KUKA KRL program: ps_603geo_x1.src, ps_603geo_x1.dat

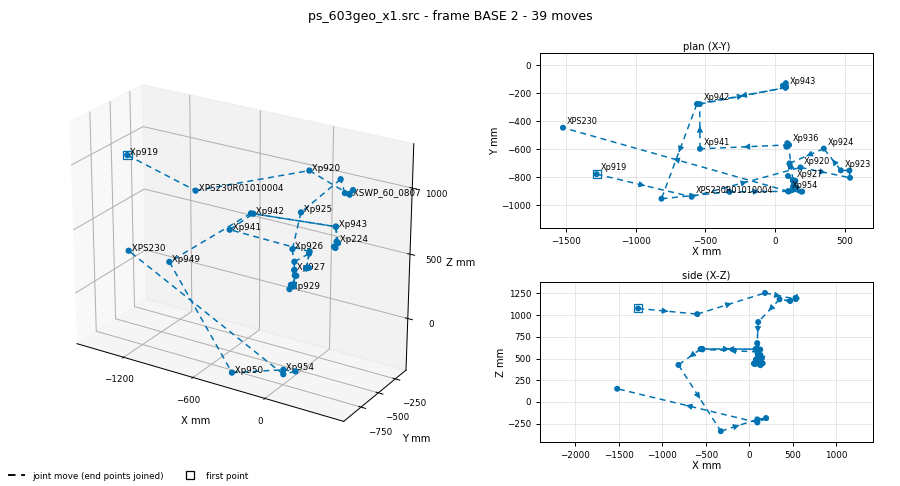
[picture p0: tool path of ps_603geo_x1.src in frame BASE 2, 39 of 39 moves have a stored position in this frame; points joined in program order, loops and branches not executed]
--- ps_603geo_x1.src ---
&ACCESS RV2
&REL 97
&COMMENT Solda Geometria x1
DEF ps_603geo_x1( )
EXT e_Fraes2 ( )
EXT f_Fraes2 ( )

  ;FOLD INI;%{PE}%V2.2.2,%MKUKATPBASIS,%CINIT,%VCOMMON,%P
  ;FOLD BAS INI;%{PE}%V2.2.2,%MKUKATPBASIS,%CINIT,%VINIT,%P
  INTERRUPT DECL 3 WHEN $STOPMESS==TRUE DO IR_STOPM ( )
  INTERRUPT ON 3
  BAS (#INITMOV,0 )
  ;ENDFOLD
  ;FOLD A20 INI;%{E}%V2.2.2,%MKUKATPA20,%CINIT,%VINIT,%P
  IF ARC20==TRUE THEN
    A20 (ARC_INI)
    INTERRUPT DECL 6 WHEN $CYCFLAG[3]==FALSE DO A20(TECH_STOP2)
  ENDIF
  ;ENDFOLD
  ;FOLD A10 INI;%{E}%V2.2.2,%MKUKATPARC,%CINIT,%VINIT,%P
  IF A10_OPTION==#ACTIVE THEN
    INTERRUPT DECL 4 WHEN $CYCFLAG[2]==FALSE DO A10 (#APPL_ERROR)
    INTERRUPT DECL 7 WHEN A_ARC_SWI==#ACTIVE DO A10 (#ARC_SEAM)
    INTERRUPT DECL 5 WHEN A_FLY_ARC==TRUE DO A10 (#HPU_ARC)
    INTERRUPT  ON 5
    A10_INI ( )
  ENDIF
  ;ENDFOLD
  ;FOLD GRIPPER INI;%{E}%V2.2.2,%MKUKATPGRIPPER,%CINIT,%VINIT,%P
  USER_GRP(0,DUMMY,DUMMY,GDEFAULT)
  ;ENDFOLD
  ;FOLD SPOT INI;%{E}%V.2.2,%MKUKATPSPOT,%CINIT,%VINIT,%P
  USERSPOT(#INIT)
  ;ENDFOLD
  ;FOLD TOUCHSENSE INI;%{E}%V2.2.2,%MKUKATPTS,%CINIT,%VINIT,%P
  IF H70_OPTION THEN
    INTERRUPT DECL 15 WHEN $MEAS_PULSE[TOUCH_I[TOUCH_ACTIVE].IN_NR] DO H70 (6,CD0 )
    INTERRUPT DECL 16 WHEN $ZERO_MOVE DO H70 (7,CD0 )
    INTERRUPT DECL 17 WHEN $TECHPAR_C[FG_TOUCH,8]>0.5 DO H70 (8,CD0)
    H70 (1,CD0 )
  ENDIF
  ;ENDFOLD
  ;FOLD USER INI;%{P}%V2.2.2,%MKUKATPUSER,%CINIT,%VINIT,%P
  ;Make your modifications here
  ;ENDFOLD
  ;ENDFOLD

; Caracterização dos meios de produção:
; Versão Atual:
; 19/07/2013 12:00 Name: P13.060-R3 CHANGES: Solda Geometria X1
; Accelo

chk_w2_wechs_ok ( )        ;VERIFICAÇÃO DE FERRAMENTA: x1

IF (NOT(GHOST())) THEN
IF MaxStandMenge(2) THEN
  MaxStandmengeErreicht(2)
ENDIF

IF Elektrodenwechsel(2) THEN
  e_Fraes2()                  ; Fresa Pinca X1
ENDIF
ENDIF

;FOLD PTP p919  Vel= 100 % P_OLP1 Tool[2]:Gun X1                   Base[2]:Accelo;%{PE}%R 4.1.16,%MKUKATPBASIS,%CMOVE,%VPTP,%P 1:PTP, 2:p919, 3:, 5:100, 7:P_OLP1
$BWDSTART = FALSE
PDAT_ACT=PP_OLP1
BAS(#PTP_DAT)
FDAT_ACT=Fp919
BAS(#FRAMES)
BAS(#VEL_PTP,100)
PTP Xp919
;ENDFOLD

;FOLD ; START INTERLOCK 2 COM R4;%{PE}%R2.2,%MKUKATPBASIS,%CCOMMENT,%VNORMAL,%P 2: START INTERLOCK 2 COM R4
;ENDFOLD
;FOLD Kollision.Ueberwachung_4_Ein ;%{PE}%MKUKATPUSER
COLLSTOP( 4, 1 ) ;INTERRUPTUEBERWACHT
;ENDFOLD

;FOLD PTP PS230R01010004 CONT Vel= 100 % PDAT3 Tool[2]:Gun X1                   Base[2]:Accelo;%{PE}%R 4.1.16,%MKUKATPBASIS,%CMOVE,%VPTP,%P 1:PTP, 2:PS230R01010004, 3:C_PTP, 5:100, 7:PDAT3
$BWDSTART = FALSE
PDAT_ACT=PPDAT3
BAS(#PTP_DAT)
FDAT_ACT=FPS230R01010004
BAS(#FRAMES)
BAS(#VEL_PTP,100)
PTP XPS230R01010004 C_PTP
;ENDFOLD

;FOLD OUT 839 'Soldando'  State= TRUE ;%{PE}%R 4.1.16,%MKUKATPBASIS,%COUT,%VOUTX,%P 2:839, 3:'Soldando', 5:TRUE, 6:
$OUT[839]=TRUE
;ENDFOLD
;FOLD OUT 848 'Area de Solda'  State= FALSE ;%{PE}%R 4.1.16,%MKUKATPBASIS,%COUT,%VOUTX,%P 2:848, 3:'Area de Solda', 5:FALSE, 6:
$OUT[848]=FALSE
;ENDFOLD

;FOLD PTP p920 CONT Vel= 100 % P_OLP2 Tool[2]:Gun X1                   Base[2]:Accelo;%{PE}%R 4.1.16,%MKUKATPBASIS,%CMOVE,%VPTP,%P 1:PTP, 2:p920, 3:C_PTP, 5:100, 7:P_OLP2
$BWDSTART = FALSE
PDAT_ACT=PP_OLP2
BAS(#PTP_DAT)
FDAT_ACT=Fp920
BAS(#FRAMES)
BAS(#VEL_PTP,100)
PTP Xp920 C_PTP
;ENDFOLD

;FOLD ; SWP_60_0807;%{PE}%R2.2,%MKUKATPBASIS,%CCOMMENT,%VNORMAL,%P 2: SWP_60_0807
;ENDFOLD
;FOLD PTP SWP_60_0807 PDAT4 SPOT Gun= 2 RETR CLS PgNo1= 121 ACTIVE= 1 Tool[2]:Gun X1                   Base[2]:Accelo;%{PE}%R 4.1.12,%MKUKATPSPOT,%CSPOT,%VPTP,%P 1:PTP, 2:SWP_60_0807, 3:, 5:100, 7:PDAT4, 10:2, 12:#FIRST, 14:#CLO, 16:121, 18:1, 20:0, 22:0, 24:1, 25:NORMAL
$BWDSTART = FALSE
PDAT_ACT=PPDAT4
BAS(#PTP_DAT)
FDAT_ACT=FSWP_60_0807
BAS(#FRAMES)
BAS(#VEL_PTP,PPDAT4.VEL)
S_ACT.GUN=2
S_ACT.PAIR=SDEFAULT.PAIR
S_ACT.RETR=#CLO
S_ACT.CLO_TM=1
S_ACT.PGNO1=121
S_ACT.PGNO2=SDEFAULT.PGNO2
S_ACT.PRESS1=SDEFAULT.PRESS1
S_ACT.PRESS2=SDEFAULT.PRESS2
S_READY=FALSE
PTP XSWP_60_0807
USERSPOT(#SPOT, S_ACT)
WAIT FOR S_READY
;ENDFOLD

;FOLD ; SWP_60_0403;%{PE}%R2.2,%MKUKATPBASIS,%CCOMMENT,%VNORMAL,%P 2: SWP_60_0403
;ENDFOLD
;FOLD PTP SWP_60_0403 PDAT5 SPOT Gun= 2 RETR OPN PgNo1= 122 ACTIVE= 1 Tool[2]:Gun X1                   Base[2]:Accelo;%{PE}%R 4.1.12,%MKUKATPSPOT,%CSPOT,%VPTP,%P 1:PTP, 2:SWP_60_0403, 3:, 5:100, 7:PDAT5, 10:2, 12:#FIRST, 14:#OPN, 16:122, 18:1, 20:0, 22:0, 24:1, 25:NORMAL
$BWDSTART = FALSE
PDAT_ACT=PPDAT5
BAS(#PTP_DAT)
FDAT_ACT=FSWP_60_0403
BAS(#FRAMES)
BAS(#VEL_PTP,PPDAT5.VEL)
S_ACT.GUN=2
S_ACT.PAIR=SDEFAULT.PAIR
S_ACT.RETR=#OPN
S_ACT.CLO_TM=1
S_ACT.PGNO1=122
S_ACT.PGNO2=SDEFAULT.PGNO2
S_ACT.PRESS1=SDEFAULT.PRESS1
S_ACT.PRESS2=SDEFAULT.PRESS2
S_READY=FALSE
PTP XSWP_60_0403
USERSPOT(#SPOT, S_ACT)
WAIT FOR S_READY
;ENDFOLD

;FOLD PTP p923 CONT Vel= 100 % P_OLP5 Tool[2]:Gun X1                   Base[2]:Accelo;%{PE}%R 4.1.16,%MKUKATPBASIS,%CMOVE,%VPTP,%P 1:PTP, 2:p923, 3:C_PTP, 5:100, 7:P_OLP5
$BWDSTART = FALSE
PDAT_ACT=PP_OLP5
BAS(#PTP_DAT)
FDAT_ACT=Fp923
BAS(#FRAMES)
BAS(#VEL_PTP,100)
PTP Xp923 C_PTP
;ENDFOLD
;FOLD PTP p924 CONT Vel= 100 % P_OLP6 Tool[2]:Gun X1                   Base[2]:Accelo;%{PE}%R 4.1.16,%MKUKATPBASIS,%CMOVE,%VPTP,%P 1:PTP, 2:p924, 3:C_PTP, 5:100, 7:P_OLP6
$BWDSTART = FALSE
PDAT_ACT=PP_OLP6
BAS(#PTP_DAT)
FDAT_ACT=Fp924
BAS(#FRAMES)
BAS(#VEL_PTP,100)
PTP Xp924 C_PTP
;ENDFOLD
;FOLD PTP p925 CONT Vel= 100 % P_OLP7 Tool[2]:Gun X1                   Base[2]:Accelo;%{PE}%R 4.1.16,%MKUKATPBASIS,%CMOVE,%VPTP,%P 1:PTP, 2:p925, 3:C_PTP, 5:100, 7:P_OLP7
$BWDSTART = FALSE
PDAT_ACT=PP_OLP7
BAS(#PTP_DAT)
FDAT_ACT=Fp925
BAS(#FRAMES)
BAS(#VEL_PTP,100)
PTP Xp925 C_PTP
;ENDFOLD
;FOLD PTP p926 CONT Vel= 100 % P_OLP8 Tool[2]:Gun X1                   Base[2]:Accelo;%{PE}%R 4.1.16,%MKUKATPBASIS,%CMOVE,%VPTP,%P 1:PTP, 2:p926, 3:C_PTP, 5:100, 7:P_OLP8
$BWDSTART = FALSE
PDAT_ACT=PP_OLP8
BAS(#PTP_DAT)
FDAT_ACT=Fp926
BAS(#FRAMES)
BAS(#VEL_PTP,100)
PTP Xp926 C_PTP
;ENDFOLD

;FOLD ; END INTERLOCK 2 COM R4;%{PE}%R2.2,%MKUKATPBASIS,%CCOMMENT,%VNORMAL,%P 2: END INTERLOCK 2 COM R4
;ENDFOLD
;FOLD Kollision.Ueberwachung_4_Aus ;%{PE}%MKUKATPUSER
COLLSTOP( 4, 2 )
;ENDFOLD

;FOLD PTP p927 CONT Vel= 100 % P_OLP9 Tool[2]:Gun X1                   Base[2]:Accelo;%{PE}%R 4.1.16,%MKUKATPBASIS,%CMOVE,%VPTP,%P 1:PTP, 2:p927, 3:C_PTP, 5:100, 7:P_OLP9
$BWDSTART = FALSE
PDAT_ACT=PP_OLP9
BAS(#PTP_DAT)
FDAT_ACT=Fp927
BAS(#FRAMES)
BAS(#VEL_PTP,100)
PTP Xp927 C_PTP
;ENDFOLD
;FOLD PTP p928 CONT Vel= 100 % P_OLP10 Tool[2]:Gun X1                   Base[2]:Accelo;%{PE}%R 4.1.16,%MKUKATPBASIS,%CMOVE,%VPTP,%P 1:PTP, 2:p928, 3:C_PTP, 5:100, 7:P_OLP10
$BWDSTART = FALSE
PDAT_ACT=PP_OLP10
BAS(#PTP_DAT)
FDAT_ACT=Fp928
BAS(#FRAMES)
BAS(#VEL_PTP,100)
PTP Xp928 C_PTP
;ENDFOLD
;FOLD PTP p929 CONT Vel= 100 % P_OLP11 Tool[2]:Gun X1                   Base[2]:Accelo;%{PE}%R 4.1.16,%MKUKATPBASIS,%CMOVE,%VPTP,%P 1:PTP, 2:p929, 3:C_PTP, 5:100, 7:P_OLP11
$BWDSTART = FALSE
PDAT_ACT=PP_OLP11
BAS(#PTP_DAT)
FDAT_ACT=Fp929
BAS(#FRAMES)
BAS(#VEL_PTP,100)
PTP Xp929 C_PTP
;ENDFOLD

;FOLD ; SWP_60_0769;%{PE}%R2.2,%MKUKATPBASIS,%CCOMMENT,%VNORMAL,%P 2: SWP_60_0769
;ENDFOLD
;FOLD PTP SWP_60_0769 PDAT6 SPOT Gun= 2 RETR OPN PgNo1= 123 ACTIVE= 1 Tool[2]:Gun X1                   Base[2]:Accelo;%{PE}%R 4.1.12,%MKUKATPSPOT,%CSPOT,%VPTP,%P 1:PTP, 2:SWP_60_0769, 3:, 5:100, 7:PDAT6, 10:2, 12:#FIRST, 14:#OPN, 16:123, 18:1, 20:0, 22:0, 24:1, 25:NORMAL
$BWDSTART = FALSE
PDAT_ACT=PPDAT6
BAS(#PTP_DAT)
FDAT_ACT=FSWP_60_0769
BAS(#FRAMES)
BAS(#VEL_PTP,PPDAT6.VEL)
S_ACT.GUN=2
S_ACT.PAIR=SDEFAULT.PAIR
S_ACT.RETR=#OPN
S_ACT.CLO_TM=1
S_ACT.PGNO1=123
S_ACT.PGNO2=SDEFAULT.PGNO2
S_ACT.PRESS1=SDEFAULT.PRESS1
S_ACT.PRESS2=SDEFAULT.PRESS2
S_READY=FALSE
PTP XSWP_60_0769
USERSPOT(#SPOT, S_ACT)
WAIT FOR S_READY
;ENDFOLD

;FOLD PTP p931 CONT Vel= 100 % P_OLP13 Tool[2]:Gun X1                   Base[2]:Accelo;%{PE}%R 4.1.16,%MKUKATPBASIS,%CMOVE,%VPTP,%P 1:PTP, 2:p931, 3:C_PTP, 5:100, 7:P_OLP13
$BWDSTART = FALSE
PDAT_ACT=PP_OLP13
BAS(#PTP_DAT)
FDAT_ACT=Fp931
BAS(#FRAMES)
BAS(#VEL_PTP,100)
PTP Xp931 C_PTP
;ENDFOLD

;FOLD ; SWP_60_0161;%{PE}%R2.2,%MKUKATPBASIS,%CCOMMENT,%VNORMAL,%P 2: SWP_60_0161
;ENDFOLD
;FOLD PTP SWP_60_0161 PDAT7 SPOT Gun= 2 RETR OPN PgNo1= 124 ACTIVE= 1 Tool[2]:Gun X1                   Base[2]:Accelo;%{PE}%R 4.1.12,%MKUKATPSPOT,%CSPOT,%VPTP,%P 1:PTP, 2:SWP_60_0161, 3:, 5:100, 7:PDAT7, 10:2, 12:#FIRST, 14:#OPN, 16:124, 18:1, 20:0, 22:0, 24:1, 25:NORMAL
$BWDSTART = FALSE
PDAT_ACT=PPDAT7
BAS(#PTP_DAT)
FDAT_ACT=FSWP_60_0161
BAS(#FRAMES)
BAS(#VEL_PTP,PPDAT7.VEL)
S_ACT.GUN=2
S_ACT.PAIR=SDEFAULT.PAIR
S_ACT.RETR=#OPN
S_ACT.CLO_TM=1
S_ACT.PGNO1=124
S_ACT.PGNO2=SDEFAULT.PGNO2
S_ACT.PRESS1=SDEFAULT.PRESS1
S_ACT.PRESS2=SDEFAULT.PRESS2
S_READY=FALSE
PTP XSWP_60_0161
USERSPOT(#SPOT, S_ACT)
WAIT FOR S_READY
;ENDFOLD

;FOLD PTP p933 CONT Vel= 100 % P_OLP15 Tool[2]:Gun X1                   Base[2]:Accelo;%{PE}%R 4.1.16,%MKUKATPBASIS,%CMOVE,%VPTP,%P 1:PTP, 2:p933, 3:C_PTP, 5:100, 7:P_OLP15
$BWDSTART = FALSE
PDAT_ACT=PP_OLP15
BAS(#PTP_DAT)
FDAT_ACT=Fp933
BAS(#FRAMES)
BAS(#VEL_PTP,100)
PTP Xp933 C_PTP
;ENDFOLD
;FOLD PTP p934 CONT Vel= 100 % P_OLP16 Tool[2]:Gun X1                   Base[2]:Accelo;%{PE}%R 4.1.16,%MKUKATPBASIS,%CMOVE,%VPTP,%P 1:PTP, 2:p934, 3:C_PTP, 5:100, 7:P_OLP16
$BWDSTART = FALSE
PDAT_ACT=PP_OLP16
BAS(#PTP_DAT)
FDAT_ACT=Fp934
BAS(#FRAMES)
BAS(#VEL_PTP,100)
PTP Xp934 C_PTP
;ENDFOLD
;FOLD PTP p935 CONT Vel= 100 % P_OLP17 Tool[2]:Gun X1                   Base[2]:Accelo;%{PE}%R 4.1.16,%MKUKATPBASIS,%CMOVE,%VPTP,%P 1:PTP, 2:p935, 3:C_PTP, 5:100, 7:P_OLP17
$BWDSTART = FALSE
PDAT_ACT=PP_OLP17
BAS(#PTP_DAT)
FDAT_ACT=Fp935
BAS(#FRAMES)
BAS(#VEL_PTP,100)
PTP Xp935 C_PTP
;ENDFOLD
;FOLD PTP p936 CONT Vel= 100 % P_OLP18 Tool[2]:Gun X1                   Base[2]:Accelo;%{PE}%R 4.1.16,%MKUKATPBASIS,%CMOVE,%VPTP,%P 1:PTP, 2:p936, 3:C_PTP, 5:100, 7:P_OLP18
$BWDSTART = FALSE
PDAT_ACT=PP_OLP18
BAS(#PTP_DAT)
FDAT_ACT=Fp936
BAS(#FRAMES)
BAS(#VEL_PTP,100)
PTP Xp936 C_PTP
;ENDFOLD
;FOLD PTP p937 CONT Vel= 100 % P_OLP19 Tool[2]:Gun X1                   Base[2]:Accelo;%{PE}%R 4.1.16,%MKUKATPBASIS,%CMOVE,%VPTP,%P 1:PTP, 2:p937, 3:C_PTP, 5:100, 7:P_OLP19
$BWDSTART = FALSE
PDAT_ACT=PP_OLP19
BAS(#PTP_DAT)
FDAT_ACT=Fp937
BAS(#FRAMES)
BAS(#VEL_PTP,100)
PTP Xp937 C_PTP
;ENDFOLD

;FOLD ; SWP_60_0151;%{PE}%R2.2,%MKUKATPBASIS,%CCOMMENT,%VNORMAL,%P 2: SWP_60_0151
;ENDFOLD
;FOLD PTP SWP_60_0151 PDAT8 SPOT Gun= 2 RETR OPN PgNo1= 125 ACTIVE= 1 Tool[2]:Gun X1                   Base[2]:Accelo;%{PE}%R 4.1.12,%MKUKATPSPOT,%CSPOT,%VPTP,%P 1:PTP, 2:SWP_60_0151, 3:, 5:100, 7:PDAT8, 10:2, 12:#FIRST, 14:#OPN, 16:125, 18:1, 20:0, 22:0, 24:1, 25:NORMAL
$BWDSTART = FALSE
PDAT_ACT=PPDAT8
BAS(#PTP_DAT)
FDAT_ACT=FSWP_60_0151
BAS(#FRAMES)
BAS(#VEL_PTP,PPDAT8.VEL)
S_ACT.GUN=2
S_ACT.PAIR=SDEFAULT.PAIR
S_ACT.RETR=#OPN
S_ACT.CLO_TM=1
S_ACT.PGNO1=125
S_ACT.PGNO2=SDEFAULT.PGNO2
S_ACT.PRESS1=SDEFAULT.PRESS1
S_ACT.PRESS2=SDEFAULT.PRESS2
S_READY=FALSE
PTP XSWP_60_0151
USERSPOT(#SPOT, S_ACT)
WAIT FOR S_READY
;ENDFOLD

;FOLD PTP p939 CONT Vel= 100 % P_OLP21 Tool[2]:Gun X1                   Base[2]:Accelo;%{PE}%R 4.1.16,%MKUKATPBASIS,%CMOVE,%VPTP,%P 1:PTP, 2:p939, 3:C_PTP, 5:100, 7:P_OLP21
$BWDSTART = FALSE
PDAT_ACT=PP_OLP21
BAS(#PTP_DAT)
FDAT_ACT=Fp939
BAS(#FRAMES)
BAS(#VEL_PTP,100)
PTP Xp939 C_PTP
;ENDFOLD
;FOLD PTP p940 CONT Vel= 100 % P_OLP22 Tool[2]:Gun X1                   Base[2]:Accelo;%{PE}%R 4.1.16,%MKUKATPBASIS,%CMOVE,%VPTP,%P 1:PTP, 2:p940, 3:C_PTP, 5:100, 7:P_OLP22
$BWDSTART = FALSE
PDAT_ACT=PP_OLP22
BAS(#PTP_DAT)
FDAT_ACT=Fp940
BAS(#FRAMES)
BAS(#VEL_PTP,100)
PTP Xp940 C_PTP
;ENDFOLD
;FOLD PTP p941  Vel= 100 % P_OLP23 Tool[2]:Gun X1                   Base[2]:Accelo;%{PE}%R 4.1.16,%MKUKATPBASIS,%CMOVE,%VPTP,%P 1:PTP, 2:p941, 3:, 5:100, 7:P_OLP23
$BWDSTART = FALSE
PDAT_ACT=PP_OLP23
BAS(#PTP_DAT)
FDAT_ACT=Fp941
BAS(#FRAMES)
BAS(#VEL_PTP,100)
PTP Xp941
;ENDFOLD

;FOLD ; START INTERLOCK 2 COM R4;%{PE}%R2.2,%MKUKATPBASIS,%CCOMMENT,%VNORMAL,%P 2: START INTERLOCK 2 COM R4
;ENDFOLD
;FOLD Kollision.Ueberwachung_4_Ein ;%{PE}%MKUKATPUSER
COLLSTOP( 4, 1 ) ;INTERRUPTUEBERWACHT
;ENDFOLD

;FOLD PTP p942 CONT Vel= 100 % P_OLP24 Tool[2]:Gun X1                   Base[2]:Accelo;%{PE}%R 4.1.16,%MKUKATPBASIS,%CMOVE,%VPTP,%P 1:PTP, 2:p942, 3:C_PTP, 5:100, 7:P_OLP24
$BWDSTART = FALSE
PDAT_ACT=PP_OLP24
BAS(#PTP_DAT)
FDAT_ACT=Fp942
BAS(#FRAMES)
BAS(#VEL_PTP,100)
PTP Xp942 C_PTP
;ENDFOLD
;FOLD PTP p943 CONT Vel= 100 % P_OLP25 Tool[2]:Gun X1                   Base[2]:Accelo;%{PE}%R 4.1.16,%MKUKATPBASIS,%CMOVE,%VPTP,%P 1:PTP, 2:p943, 3:C_PTP, 5:100, 7:P_OLP25
$BWDSTART = FALSE
PDAT_ACT=PP_OLP25
BAS(#PTP_DAT)
FDAT_ACT=Fp943
BAS(#FRAMES)
BAS(#VEL_PTP,100)
PTP Xp943 C_PTP
;ENDFOLD
;FOLD PTP p224 CONT Vel= 100 % PDAT16 Tool[2]:Gun X1                   Base[2]:Accelo;%{PE}%R 4.1.16,%MKUKATPBASIS,%CMOVE,%VPTP,%P 1:PTP, 2:p224, 3:C_PTP, 5:100, 7:PDAT16
$BWDSTART = FALSE
PDAT_ACT=PPDAT16
BAS(#PTP_DAT)
FDAT_ACT=Fp224
BAS(#FRAMES)
BAS(#VEL_PTP,100)
PTP Xp224 C_PTP
;ENDFOLD
;FOLD PTP p944 CONT Vel= 100 % P_OLP26 Tool[2]:Gun X1                   Base[2]:Accelo;%{PE}%R 4.1.16,%MKUKATPBASIS,%CMOVE,%VPTP,%P 1:PTP, 2:p944, 3:C_PTP, 5:100, 7:P_OLP26
$BWDSTART = FALSE
PDAT_ACT=PP_OLP26
BAS(#PTP_DAT)
FDAT_ACT=Fp944
BAS(#FRAMES)
BAS(#VEL_PTP,100)
PTP Xp944 C_PTP
;ENDFOLD

;FOLD ; SWP_60_0133;%{PE}%R2.2,%MKUKATPBASIS,%CCOMMENT,%VNORMAL,%P 2: SWP_60_0133
;ENDFOLD
;FOLD PTP SWP_60_0133 PDAT9 SPOT Gun= 2 RETR OPN PgNo1= 126 ACTIVE= 1 Tool[2]:Gun X1                   Base[2]:Accelo;%{PE}%R 4.1.12,%MKUKATPSPOT,%CSPOT,%VPTP,%P 1:PTP, 2:SWP_60_0133, 3:, 5:100, 7:PDAT9, 10:2, 12:#FIRST, 14:#OPN, 16:126, 18:1, 20:0, 22:0, 24:1, 25:NORMAL
$BWDSTART = FALSE
PDAT_ACT=PPDAT9
BAS(#PTP_DAT)
FDAT_ACT=FSWP_60_0133
BAS(#FRAMES)
BAS(#VEL_PTP,PPDAT9.VEL)
S_ACT.GUN=2
S_ACT.PAIR=SDEFAULT.PAIR
S_ACT.RETR=#OPN
S_ACT.CLO_TM=1
S_ACT.PGNO1=126
S_ACT.PGNO2=SDEFAULT.PGNO2
S_ACT.PRESS1=SDEFAULT.PRESS1
S_ACT.PRESS2=SDEFAULT.PRESS2
S_READY=FALSE
PTP XSWP_60_0133
USERSPOT(#SPOT, S_ACT)
WAIT FOR S_READY
;ENDFOLD

;FOLD PTP p946  Vel= 100 % P_OLP28 Tool[2]:Gun X1                   Base[2]:Accelo;%{PE}%R 4.1.16,%MKUKATPBASIS,%CMOVE,%VPTP,%P 1:PTP, 2:p946, 3:, 5:100, 7:P_OLP28
$BWDSTART = FALSE
PDAT_ACT=PP_OLP28
BAS(#PTP_DAT)
FDAT_ACT=Fp946
BAS(#FRAMES)
BAS(#VEL_PTP,100)
PTP Xp946
;ENDFOLD

;FOLD PTP p225 CONT Vel= 100 % PDAT17 Tool[2]:Gun X1                   Base[2]:Accelo;%{PE}%R 4.1.16,%MKUKATPBASIS,%CMOVE,%VPTP,%P 1:PTP, 2:p225, 3:C_PTP, 5:100, 7:PDAT17
$BWDSTART = FALSE
PDAT_ACT=PPDAT17
BAS(#PTP_DAT)
FDAT_ACT=Fp225
BAS(#FRAMES)
BAS(#VEL_PTP,100)
PTP Xp225 C_PTP
;ENDFOLD
;FOLD PTP p947 CONT Vel= 100 % P_OLP29 Tool[2]:Gun X1                   Base[2]:Accelo;%{PE}%R 4.1.16,%MKUKATPBASIS,%CMOVE,%VPTP,%P 1:PTP, 2:p947, 3:C_PTP, 5:100, 7:P_OLP29
$BWDSTART = FALSE
PDAT_ACT=PP_OLP29
BAS(#PTP_DAT)
FDAT_ACT=Fp947
BAS(#FRAMES)
BAS(#VEL_PTP,100)
PTP Xp947 C_PTP
;ENDFOLD
;FOLD PTP p948 CONT Vel= 100 % P_OLP30 Tool[2]:Gun X1                   Base[2]:Accelo;%{PE}%R 4.1.16,%MKUKATPBASIS,%CMOVE,%VPTP,%P 1:PTP, 2:p948, 3:C_PTP, 5:100, 7:P_OLP30
$BWDSTART = FALSE
PDAT_ACT=PP_OLP30
BAS(#PTP_DAT)
FDAT_ACT=Fp948
BAS(#FRAMES)
BAS(#VEL_PTP,100)
PTP Xp948 C_PTP
;ENDFOLD
;FOLD PTP p949 CONT Vel= 100 % P_OLP31 Tool[2]:Gun X1                   Base[2]:Accelo;%{PE}%R 4.1.16,%MKUKATPBASIS,%CMOVE,%VPTP,%P 1:PTP, 2:p949, 3:C_PTP, 5:100, 7:P_OLP31
$BWDSTART = FALSE
PDAT_ACT=PP_OLP31
BAS(#PTP_DAT)
FDAT_ACT=Fp949
BAS(#FRAMES)
BAS(#VEL_PTP,100)
PTP Xp949 C_PTP
;ENDFOLD
;FOLD PTP p950 CONT Vel= 100 % P_OLP32 Tool[2]:Gun X1                   Base[2]:Accelo;%{PE}%R 4.1.16,%MKUKATPBASIS,%CMOVE,%VPTP,%P 1:PTP, 2:p950, 3:C_PTP, 5:100, 7:P_OLP32
$BWDSTART = FALSE
PDAT_ACT=PP_OLP32
BAS(#PTP_DAT)
FDAT_ACT=Fp950
BAS(#FRAMES)
BAS(#VEL_PTP,100)
PTP Xp950 C_PTP
;ENDFOLD
;FOLD PTP p954 CONT Vel= 100 % P_OLP36 Tool[2]:Gun X1                   Base[2]:Accelo;%{PE}%R 4.1.16,%MKUKATPBASIS,%CMOVE,%VPTP,%P 1:PTP, 2:p954, 3:C_PTP, 5:100, 7:P_OLP36
$BWDSTART = FALSE
PDAT_ACT=PP_OLP36
BAS(#PTP_DAT)
FDAT_ACT=Fp954
BAS(#FRAMES)
BAS(#VEL_PTP,100)
PTP Xp954 C_PTP
;ENDFOLD

;FOLD ; SWP_60_0443;%{PE}%R2.2,%MKUKATPBASIS,%CCOMMENT,%VNORMAL,%P 2: SWP_60_0443
;ENDFOLD
;FOLD PTP SWP_60_0443 PDAT11 SPOT Gun= 2 RETR CLS PgNo1= 128 ACTIVE= 1 Tool[2]:Gun X1                   Base[2]:Accelo;%{PE}%R 4.1.12,%MKUKATPSPOT,%CSPOT,%VPTP,%P 1:PTP, 2:SWP_60_0443, 3:, 5:100, 7:PDAT11, 10:2, 12:#FIRST, 14:#CLO, 16:128, 18:1, 20:0, 22:0, 24:1, 25:NORMAL
$BWDSTART = FALSE
PDAT_ACT=PPDAT11
BAS(#PTP_DAT)
FDAT_ACT=FSWP_60_0443
BAS(#FRAMES)
BAS(#VEL_PTP,PPDAT11.VEL)
S_ACT.GUN=2
S_ACT.PAIR=SDEFAULT.PAIR
S_ACT.RETR=#CLO
S_ACT.CLO_TM=1
S_ACT.PGNO1=128
S_ACT.PGNO2=SDEFAULT.PGNO2
S_ACT.PRESS1=SDEFAULT.PRESS1
S_ACT.PRESS2=SDEFAULT.PRESS2
S_READY=FALSE
PTP XSWP_60_0443
USERSPOT(#SPOT, S_ACT)
WAIT FOR S_READY
;ENDFOLD

;FOLD PTP p960 CONT Vel= 100 % P_OLP42 Tool[2]:Gun X1                   Base[2]:Accelo;%{PE}%R 4.1.16,%MKUKATPBASIS,%CMOVE,%VPTP,%P 1:PTP, 2:p960, 3:C_PTP, 5:100, 7:P_OLP42
$BWDSTART = FALSE
PDAT_ACT=PP_OLP42
BAS(#PTP_DAT)
FDAT_ACT=Fp960
BAS(#FRAMES)
BAS(#VEL_PTP,100)
PTP Xp960 C_PTP
;ENDFOLD

;FOLD OUT 839 'Soldando'  State= FALSE ;%{PE}%R 4.1.16,%MKUKATPBASIS,%COUT,%VOUTX,%P 2:839, 3:'Soldando', 5:FALSE, 6:
$OUT[839]=FALSE
;ENDFOLD
;FOLD OUT 848 'Area de Solda'  State= TRUE ;%{PE}%R 4.1.16,%MKUKATPBASIS,%COUT,%VOUTX,%P 2:848, 3:'Area de Solda', 5:TRUE, 6:
$OUT[848]=TRUE
;ENDFOLD

;FOLD PTP PS230  Vel= 100 % PDAT2 Tool[2]:Gun X1                   Base[2]:Accelo;%{PE}%R 4.1.16,%MKUKATPBASIS,%CMOVE,%VPTP,%P 1:PTP, 2:PS230, 3:, 5:100, 7:PDAT2
$BWDSTART = FALSE
PDAT_ACT=PPDAT2
BAS(#PTP_DAT)
FDAT_ACT=FPS230
BAS(#FRAMES)
BAS(#VEL_PTP,100)
PTP XPS230
;ENDFOLD

;FOLD ; END  INTERLOCK 2 COM R4;%{PE}%R 4.1.16,%MKUKATPBASIS,%CCOMMENT,%VNORMAL,%P 2:END  INTERLOCK 2 COM R4
;ENDFOLD
;FOLD Kollision.Ueberwachung_4_Aus ;%{PE}%MKUKATPUSER
COLLSTOP( 4, 2 )
;ENDFOLD

;FOLD OUT 840 'Solda Geometria Concluida'  State= TRUE CONT;%{PE}%R 4.1.16,%MKUKATPBASIS,%COUT,%VOUTX,%P 2:840, 3:'Solda Geometria Concluida', 5:TRUE, 6:CONTINUE
CONTINUE
$OUT[840]=TRUE
;ENDFOLD
;FOLD OUT 837 'Solic. Lib. Soldar Respot GEO 2'  State= TRUE ;%{PE}%R 4.1.16,%MKUKATPBASIS,%COUT,%VOUTX,%P 2:837, 3:'Solic. Lib. Soldar Respot GEO 2', 5:TRUE, 6:
$OUT[837]=TRUE
;ENDFOLD
;FOLD WAIT Time= 0.7 sec;%{PE}%R 4.1.16,%MKUKATPBASIS,%CWAIT,%VWAIT,%P 2:0.7
WAIT SEC 0.7
;ENDFOLD
;FOLD OUT 840 'Solda Geometria Concluida'  State= FALSE CONT;%{PE}%R 4.1.16,%MKUKATPBASIS,%COUT,%VOUTX,%P 2:840, 3:'Solda Geometria Concluida', 5:FALSE, 6:CONTINUE
CONTINUE
$OUT[840]=FALSE
;ENDFOLD

end_weld_respot()     ;Fim Solda Respot

IF(NOT(GHOST())) THEN
IF FraesAnf(2) THEN
  f_Fraes2()           ; Fresa Pinca X1
ENDIF
ENDIF

END

--- ps_603geo_x1.dat ---
&ACCESS RV2
&REL 97
&COMMENT Solda Geometria x1
DEFDAT  PS_603GEO_X1
;FOLD EXTERNAL DECLARATIONS;%{PE}%V2.2.2,%MKUKATPBASIS,%CEXT,%VCOMMON,%P
;FOLD BAS EXT;%{PE}%V2.2.2,%MKUKATPBASIS,%CEXT,%VEXT,%P
EXT  BAS (BAS_COMMAND  :IN,REAL  :IN )
DECL INT SUCCESS
;ENDFOLD
;FOLD A10 EXT;%{E}%V2.2.2,%MKUKATPARC,%CEXT,%VEXT,%P
EXT  A10 (A_CMD_T  :IN,A_STRT_T  :IN,A_WELD_T  :IN,A_END_T  :IN,INT  :IN )
;ENDFOLD
;FOLD A20 EXT;%{E}%V2.2.2,%MKUKATPA20,%CEXT,%VEXT,%P
EXT  A20 (INT  :IN,WELD_ST  :IN,WELD_FI  :IN,INT  :IN )
;ENDFOLD
;FOLD GRIPPER EXT;%{E}%V2.2.2,%MKUKATPGRIPPER,%CEXT,%VEXT,%P
EXT  H50 (INT  :IN,INT  :IN,INT  :IN,GRP_TYP  :IN )
;ENDFOLD
;FOLD SPOT EXT;%{E}%V2.2.2,%MKUKATPSPOT,%CEXT,%VEXT,%P
EXT  USERSPOT (S_COMMAND  :IN,SPOT_TYPE  :IN )
;ENDFOLD
;FOLD TOUCHSENSE EXT;%{E}%V2.2.2,%MKUKATPTS,%CEXT,%VEXT,%P
EXT  H70 (INT  :IN,SRCH_TYP_2  :OUT,E6POS  :IN,SRCH_TYP_3  :IN,SRCH_TYP_2  :IN,SRCH_TYP_2  :IN,SRCH_TYP_2  :IN,SRCH_TYP_2  :IN,SRCH_TYP_2  :IN,INT  :IN )
;ENDFOLD
;FOLD USER EXT;%{}%V2.2.2,%MKUKATPUSER,%CEXT,%VEXT,%P
;Make here your modifications
;ENDFOLD
;ENDFOLD

;# ============ START PATH : swp_p13060r3_ltc_geo_x1 =============
DECL FDAT Fp919={TOOL_NO 2,BASE_NO 2,IPO_FRAME #BASE}
DECL PDAT PP_OLP1={VEL 100.0,ACC 100.0,APO_DIST 40.0}
DECL E6POS Xp919={x -1278.44702,y -779.18573,z 1075.55701,a 12.3480396,b -25.9995003,c -156.968704,s 2,t 35,e1 0.0,e2 0.0,e3 0.0,e4 0.0,e5 0.0,e6 0.0}
DECL FDAT Fp920={TOOL_NO 2,BASE_NO 2,IPO_FRAME #BASE}
DECL PDAT PP_OLP2={VEL 100.0,ACC 100.0,APO_DIST 100.0}
DECL E6POS Xp920={x 180.633102,y -730.699585,z 1253.87305,a -51.0044098,b -24.0758209,c -122.426102,s 2,t 34,e1 0.0,e2 0.0,e3 0.0,e4 0.0,e5 0.0,e6 0.0}
DECL FDAT Fp923={TOOL_NO 2,BASE_NO 2,IPO_FRAME #BASE}
DECL PDAT PP_OLP5={VEL 100.0,ACC 100.0,APO_DIST 100.0}
DECL E6POS Xp923={x 469.447601,y -752.146179,z 1160.90601,a -58.1620102,b -30.9620991,c -127.948601,s 2,t 34,e1 0.0,e2 0.0,e3 0.0,e4 0.0,e5 0.0,e6 0.0}
DECL FDAT Fp924={TOOL_NO 2,BASE_NO 2,IPO_FRAME #BASE}
DECL PDAT PP_OLP6={VEL 100.0,ACC 100.0,APO_DIST 100.0}
DECL E6POS Xp924={x 347.623993,y -596.088989,z 1180.43396,a -54.9714012,b -26.2077999,c -124.309502,s 2,t 34}
DECL FDAT Fp925={TOOL_NO 2,BASE_NO 2,IPO_FRAME #BASE}
DECL PDAT PP_OLP7={VEL 100.0,ACC 100.0,APO_DIST 100.0}
DECL E6POS Xp925={x 102.325996,y -701.732971,z 919.525024,a -37.8620987,b 38.7346992,c -71.782402,s 2,t 34}
DECL FDAT Fp926={TOOL_NO 2,BASE_NO 2,IPO_FRAME #BASE}
DECL PDAT PP_OLP8={VEL 100.0,ACC 100.0,APO_DIST 100.0}
DECL E6POS Xp926={x 91.4629974,y -792.432983,z 677.267029,a -50.3600998,b 54.4105988,c -80.490097,s 2,t 34}
DECL FDAT Fp927={TOOL_NO 2,BASE_NO 2,IPO_FRAME #BASE}
DECL PDAT PP_OLP9={VEL 100.0,ACC 100.0,APO_DIST 100.0}
DECL E6POS Xp927={x 126.247002,y -823.231018,z 539.911987,a -41.5237007,b 71.3117981,c -72.5373001,s 2,t 34}
DECL FDAT Fp928={TOOL_NO 2,BASE_NO 2,IPO_FRAME #BASE}
DECL PDAT PP_OLP10={VEL 100.0,ACC 100.0,APO_DIST 100.0}
DECL E6POS Xp928={x 144.522995,y -827.087219,z 503.081207,a -83.4802094,b 58.4450912,c -109.187798,s 2,t 34,e1 0.0,e2 0.0,e3 0.0,e4 0.0,e5 0.0,e6 0.0}
DECL FDAT Fp929={TOOL_NO 2,BASE_NO 2,IPO_FRAME #BASE}
DECL PDAT PP_OLP11={VEL 100.0,ACC 100.0,APO_DIST 100.0}
DECL E6POS Xp929={x 127.889999,y -888.40802,z 422.569,a -83.4804001,b 58.4446983,c -109.187798,s 2,t 34}
DECL FDAT Fp931={TOOL_NO 2,BASE_NO 2,IPO_FRAME #BASE}
DECL PDAT PP_OLP13={VEL 100.0,ACC 100.0,APO_DIST 100.0}
DECL E6POS Xp931={x 127.041,y -867.892029,z 446.539001,a -97.3261032,b 57.3554993,c -119.183899,s 2,t 34}
DECL FDAT Fp933={TOOL_NO 2,BASE_NO 2,IPO_FRAME #BASE}
DECL PDAT PP_OLP15={VEL 100.0,ACC 100.0,APO_DIST 100.0}
DECL E6POS Xp933={x 135.123001,y -831.085022,z 504.863007,a -83.4802017,b 58.4449997,c -109.187798,s 2,t 34}
DECL FDAT Fp934={TOOL_NO 2,BASE_NO 2,IPO_FRAME #BASE}
DECL PDAT PP_OLP16={VEL 100.0,ACC 100.0,APO_DIST 100.0}
DECL E6POS Xp934={x 126.247002,y -823.231018,z 539.911987,a -41.5237007,b 71.3117981,c -72.5373001,s 2,t 34}
DECL FDAT Fp935={TOOL_NO 2,BASE_NO 2,IPO_FRAME #BASE}
DECL PDAT PP_OLP17={VEL 100.0,ACC 100.0,APO_DIST 100.0}
DECL E6POS Xp935={x 126.248001,y -823.22998,z 602.909973,a -41.5245018,b 71.3115997,c -72.538002,s 2,t 34}
DECL FDAT Fp936={TOOL_NO 2,BASE_NO 2,IPO_FRAME #BASE}
DECL PDAT PP_OLP18={VEL 100.0,ACC 100.0,APO_DIST 100.0}
DECL E6POS Xp936={x 95.3696289,y -570.964417,z 560.64502,a -118.056801,b 84.4840012,c -122.064598,s 2,t 34,e1 0.0,e2 0.0,e3 0.0,e4 0.0,e5 0.0,e6 0.0}
DECL FDAT Fp937={TOOL_NO 2,BASE_NO 2,IPO_FRAME #BASE}
DECL PDAT PP_OLP19={VEL 100.0,ACC 100.0,APO_DIST 100.0}
DECL E6POS Xp937={x 80.9960022,y -581.158997,z 448.753998,a -155.764999,b 76.6326981,c -159.379395,s 2,t 34}
DECL FDAT Fp939={TOOL_NO 2,BASE_NO 2,IPO_FRAME #BASE}
DECL PDAT PP_OLP21={VEL 100.0,ACC 100.0,APO_DIST 100.0}
DECL E6POS Xp939={x 80.9960022,y -581.158997,z 448.753998,a -155.764999,b 76.6326981,c -159.379395,s 2,t 34}
DECL FDAT Fp940={TOOL_NO 2,BASE_NO 2,IPO_FRAME #BASE}
DECL PDAT PP_OLP22={VEL 100.0,ACC 100.0,APO_DIST 100.0}
DECL E6POS Xp940={x 98.4520035,y -569.473999,z 576.083008,a -118.130302,b 84.4822998,c -122.137901,s 2,t 34}
DECL FDAT Fp941={TOOL_NO 2,BASE_NO 2,IPO_FRAME #BASE}
DECL PDAT PP_OLP23={VEL 100.0,ACC 100.0,APO_DIST 100.0}
DECL E6POS Xp941={x -538.595825,y -597.655029,z 604.745789,a -113.764099,b 84.4951401,c -120.625603,s 2,t 34,e1 0.0,e2 0.0,e3 0.0,e4 0.0,e5 0.0,e6 0.0}
DECL FDAT Fp942={TOOL_NO 2,BASE_NO 2,IPO_FRAME #BASE}
DECL PDAT PP_OLP24={VEL 100.0,ACC 100.0,APO_DIST 100.0}
DECL E6POS Xp942={x -540.650513,y -277.639313,z 610.718689,a -113.748802,b 84.4967422,c -120.610199,s 2,t 34,e1 0.0,e2 0.0,e3 0.0,e4 0.0,e5 0.0,e6 0.0}
DECL FDAT Fp943={TOOL_NO 2,BASE_NO 2,IPO_FRAME #BASE}
DECL PDAT PP_OLP25={VEL 100.0,ACC 100.0,APO_DIST 100.0}
DECL E6POS Xp943={x 73.5279999,y -159.830002,z 607.299011,a 78.6467972,b 70.6716995,c 81.9641037,s 2,t 34}
DECL FDAT Fp944={TOOL_NO 2,BASE_NO 2,IPO_FRAME #BASE}
DECL PDAT PP_OLP26={VEL 100.0,ACC 100.0,APO_DIST 10.0}
DECL E6POS Xp944={x 55.3050003,y -146.901993,z 442.296997,a 117.490898,b 67.3528976,c 121.1427,s 2,t 34}
DECL FDAT Fp946={TOOL_NO 2,BASE_NO 2,IPO_FRAME #BASE}
DECL PDAT PP_OLP28={VEL 100.0,ACC 100.0,APO_DIST 100.0}
DECL E6POS Xp946={x 55.3050003,y -146.901993,z 442.296997,a 117.490898,b 67.3528976,c 121.1427,s 2,t 34}
DECL FDAT Fp947={TOOL_NO 2,BASE_NO 2,IPO_FRAME #BASE}
DECL PDAT PP_OLP29={VEL 100.0,ACC 100.0,APO_DIST 100.0}
DECL E6POS Xp947={x 73.5279999,y -159.830002,z 607.299011,a 78.6467972,b 70.6716995,c 81.9641037,s 2,t 34}
DECL FDAT Fp948={TOOL_NO 2,BASE_NO 2,IPO_FRAME #BASE}
DECL PDAT PP_OLP30={VEL 100.0,ACC 100.0,APO_DIST 10.0}
DECL E6POS Xp948={x -560.521606,y -276.747498,z 608.67218,a -113.764099,b 84.4958115,c -120.626198,s 2,t 34,e1 0.0,e2 0.0,e3 0.0,e4 0.0,e5 0.0,e6 0.0}
DECL FDAT Fp949={TOOL_NO 2,BASE_NO 2,IPO_FRAME #BASE}
DECL PDAT PP_OLP31={VEL 100.0,ACC 100.0,APO_DIST 100.0}
DECL E6POS Xp949={x -814.507019,y -954.971985,z 426.325989,a -69.2182007,b -6.35389996,c -147.227905,s 2,t 35}
DECL FDAT Fp950={TOOL_NO 2,BASE_NO 2,IPO_FRAME #BASE}
DECL PDAT PP_OLP32={VEL 100.0,ACC 100.0,APO_DIST 100.0}
DECL E6POS Xp950={x -327.606995,y -905.784973,z -335.885986,a -1.99380004,b -24.7444992,c 98.453598,s 2,t 34}
DECL FDAT Fp954={TOOL_NO 2,BASE_NO 2,IPO_FRAME #BASE}
DECL PDAT PP_OLP36={VEL 100.0,ACC 100.0,APO_DIST 100.0}
DECL E6POS Xp954={x 92.8980026,y -902.103027,z -200.399994,a 0.0,b 0.0,c 90.0,s 2,t 2}
DECL FDAT Fp960={TOOL_NO 2,BASE_NO 2,IPO_FRAME #BASE}
DECL PDAT PP_OLP42={VEL 100.0,ACC 100.0,APO_DIST 100.0}
DECL E6POS Xp960={x 92.8968887,y -901.611572,z -235.684998,a 0.00029849459,b 0.000739926996,c 89.9991302,s 2,t 2,e1 0.0,e2 0.0,e3 0.0,e4 0.0,e5 0.0,e6 0.0}
DECL SPOT_SUGG_T LAST_SPOT={GUN[] "1                       ",RETR_CMD[] "#OPN                    ",CHOISE[] "#FIRST                  ",CLO_TM[] "1                       ",PGNO1[] "1                       ",PRESS1[] "0                       ",PGNO2[] "1                       ",PRESS2[] "0                       ",SPOT_PARAMS[] "NORMAL                  "}
DECL BASIS_SUGG_T LAST_BASIS={POINT1[] "p226                    ",POINT2[] "p226                    ",CP_PARAMS[] "CPDAT0                  ",PTP_PARAMS[] "PDAT18                  ",CONT[] "                        ",CP_VEL[] "2.0                     ",PTP_VEL[] "70                      "}
DECL PDAT PPDAT2={VEL 100.0,ACC 100.0,APO_DIST 10.0}
DECL E6POS XPS230R01010004={x -598.462219,y -941.111694,z 1010.35999,a -0.0718464777,b -25.7052307,c -170.060196,s 2,t 2,e1 0.0,e2 0.0,e3 0.0,e4 0.0,e5 0.0,e6 0.0}
DECL FDAT FPS230R01010004={TOOL_NO 2,BASE_NO 2,IPO_FRAME #BASE}
DECL PDAT PPDAT3={VEL 100.0,ACC 100.0,APO_DIST 100.0}
DECL E6POS XSWP_60_0807={x 535.38501,y -804.914307,z 1182.64404,a -56.7119102,b -26.6843491,c -126.135498,s 2,t 34,e1 0.0,e2 0.0,e3 0.0,e4 0.0,e5 0.0,e6 0.0}
DECL FDAT FSWP_60_0807={TOOL_NO 2,BASE_NO 2,IPO_FRAME #BASE}
DECL PDAT PPDAT4={VEL 100.0,ACC 100.0,APO_DIST 100.0}
DECL E6POS XSWP_60_0403={x 531.099609,y -753.027893,z 1196.18506,a -56.547081,b -32.6911507,c -128.814606,s 2,t 34,e1 0.0,e2 0.0,e3 0.0,e4 0.0,e5 0.0,e6 0.0}
DECL FDAT FSWP_60_0403={TOOL_NO 2,BASE_NO 2,IPO_FRAME #BASE}
DECL PDAT PPDAT5={VEL 100.0,ACC 100.0,APO_DIST 100.0}
DECL E6POS XSWP_60_0769={x 153.808701,y -875.962524,z 444.689789,a -85.3789291,b 58.4413109,c -109.144402,s 2,t 34,e1 0.0,e2 0.0,e3 0.0,e4 0.0,e5 0.0,e6 0.0}
DECL FDAT FSWP_60_0769={TOOL_NO 2,BASE_NO 2,IPO_FRAME #BASE}
DECL PDAT PPDAT6={VEL 100.0,ACC 100.0,APO_DIST 100.0}
DECL E6POS XSWP_60_0161={x 134.449905,y -842.878601,z 443.051086,a -103.979897,b 56.3225899,c -125.571098,s 2,t 34,e1 0.0,e2 0.0,e3 0.0,e4 0.0,e5 0.0,e6 0.0}
DECL FDAT FSWP_60_0161={TOOL_NO 2,BASE_NO 2,IPO_FRAME #BASE}
DECL PDAT PPDAT7={VEL 100.0,ACC 100.0,APO_DIST 100.0}
DECL E6POS XSWP_60_0151={x 86.3240433,y -557.457214,z 444.992401,a -160.241898,b 72.6341095,c -167.420303,s 2,t 34,e1 0.0,e2 0.0,e3 0.0,e4 0.0,e5 0.0,e6 0.0}
DECL FDAT FSWP_60_0151={TOOL_NO 2,BASE_NO 2,IPO_FRAME #BASE}
DECL PDAT PPDAT8={VEL 100.0,ACC 100.0,APO_DIST 100.0}
DECL E6POS XSWP_60_0133={x 65.8852234,y -146.705704,z 435.706909,a 123.145897,b 57.1310501,c 126.371597,s 2,t 34,e1 0.0,e2 0.0,e3 0.0,e4 0.0,e5 0.0,e6 0.0}
DECL FDAT FSWP_60_0133={TOOL_NO 2,BASE_NO 2,IPO_FRAME #BASE}
DECL PDAT PPDAT9={VEL 100.0,ACC 100.0,APO_DIST 100.0}
DECL E6POS XSWP_60_0443={x 192.735703,y -904.212585,z -184.863403,a 0.00449669315,b 0.0198047701,c 90.052063,s 2,t 2,e1 0.0,e2 0.0,e3 0.0,e4 0.0,e5 0.0,e6 0.0}
DECL FDAT FSWP_60_0443={TOOL_NO 2,BASE_NO 2,IPO_FRAME #BASE}
DECL PDAT PPDAT11={VEL 100.0,ACC 100.0,APO_DIST 100.0}
DECL E6POS XP224={x 77.8080597,y -153.861801,z 490.726196,a 108.635902,b 69.255249,c 112.338097,s 2,t 34,e1 0.0,e2 0.0,e3 0.0,e4 0.0,e5 0.0,e6 0.0}
DECL FDAT Fp224={TOOL_NO 2,BASE_NO 2,IPO_FRAME #BASE}
DECL PDAT PPDAT16={VEL 100.0,ACC 100.0,APO_DIST 10.0}
DECL E6POS XP225={x 75.6939697,y -127.679497,z 468.644287,a 112.888397,b 68.4357071,c 116.675003,s 2,t 34,e1 0.0,e2 0.0,e3 0.0,e4 0.0,e5 0.0,e6 0.0}
DECL FDAT Fp225={TOOL_NO 2,BASE_NO 2,IPO_FRAME #BASE}
DECL PDAT PPDAT17={VEL 100.0,ACC 100.0,APO_DIST 10.0}
DECL E6POS XPS230={x -1519.44202,y -446.458405,z 152.208603,a 55.3340607,b -2.62300491,c 121.304901,s 2,t 3,e1 0.0,e2 0.0,e3 0.0,e4 0.0,e5 0.0,e6 0.0}
DECL FDAT FPS230={TOOL_NO 2,BASE_NO 2,IPO_FRAME #BASE}
ENDDAT
